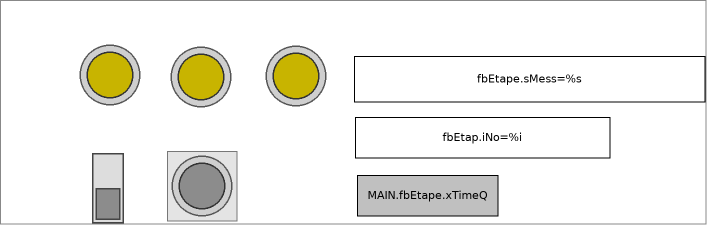
VISUALIZATION Visualization  // 707x225
    Lamp1 (75,40 70x70), variable: MAIN.QxLampe1, style: Lamp-Lamp1-Yellow
    Lamp1 (166,42 70x70), variable: MAIN.QxLampe2, style: Lamp-Lamp1-Yellow
    Lamp1 (261,41 70x70), variable: MAIN.QxLampe3, style: Lamp-Lamp1-Yellow
    DipSwitch (73,153 70x70), variable: GVL.xModePasAPas, behaviour: TOGGLE, style: Switch-DipSwitch-Gray
    PushSwitch (167,151 70x70), variable: GVL.xNextPas, behaviour: TOGGLE, style: Switch-PushSwitch-Gray
    RoundedRectangle (354,56 351x46), "fbEtape.sMess=%s", text variable: MAIN.fbEtape.sMess
    RoundedRectangle (355,117 255x41), "fbEtap.iNo=%i", text variable: MAIN.fbEtape.iNo
    RoundedRectangle (357,175 141x41), "MAIN.fbEtape.xTimeQ", colour toggle: MAIN.fbEtape.xTimeQ
END_VISUALIZATION

(* stored: Version 1.1.0.1, ProductVersion 3.1.4020.6
   Visu Visualization: Id {a1969ca4-b0e3-437c-8274-25631d0910ee} *)
